{attribute 'qualified_only'}
{attribute 'strict'}
TYPE E_InvType :
(
	brak,
	Schneider,
	ParkerAC10s
);
END_TYPE

(* stored: Version 1.1.0.1, ProductVersion 3.1.4024.15
   DUT E_InvType: Id {9359416a-6ca1-484f-a36e-83d5913bc2de} *)
